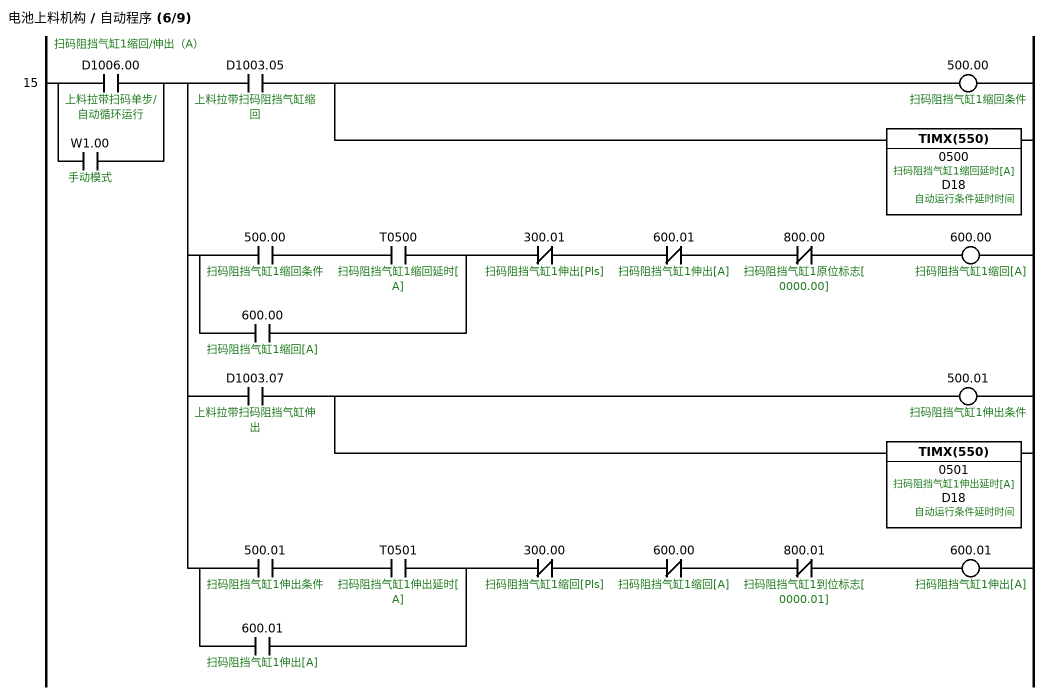
; [picture p24: 电池上料机构 / 自动程序, rungs 15-15]
; rung 15: 扫码阻挡气缸1缩回/伸出（A）
LD D1006.00  ; 上料拉带扫码单步/自动循环运行
OR W1.00  ; 手动模式
OUT TR0
AND D1003.05  ; 上料拉带扫码阻挡气缸缩回
OUT 500.00  ; 扫码阻挡气缸1缩回条件
TIMX(550) 0500 D18  ; 自动运行条件延时时间, 扫码阻挡气缸1缩回延时[A]
LD TR0
LD 500.00  ; 扫码阻挡气缸1缩回条件
AND T0500  ; 扫码阻挡气缸1缩回延时[A]
OR 600.00  ; 扫码阻挡气缸1缩回[A]
ANDLD
ANDNOT 300.01  ; 扫码阻挡气缸1伸出[Pls]
ANDNOT 600.01  ; 扫码阻挡气缸1伸出[A]
ANDNOT 800.00  ; 扫码阻挡气缸1原位标志[0000.00]
OUT 600.00  ; 扫码阻挡气缸1缩回[A]
LD TR0
AND D1003.07  ; 上料拉带扫码阻挡气缸伸出
OUT 500.01  ; 扫码阻挡气缸1伸出条件
TIMX(550) 0501 D18  ; 自动运行条件延时时间, 扫码阻挡气缸1伸出延时[A]
LD TR0
LD 500.01  ; 扫码阻挡气缸1伸出条件
AND T0501  ; 扫码阻挡气缸1伸出延时[A]
OR 600.01  ; 扫码阻挡气缸1伸出[A]
ANDLD
ANDNOT 300.00  ; 扫码阻挡气缸1缩回[Pls]
ANDNOT 600.00  ; 扫码阻挡气缸1缩回[A]
ANDNOT 800.01  ; 扫码阻挡气缸1到位标志[0000.01]
OUT 600.01  ; 扫码阻挡气缸1伸出[A]

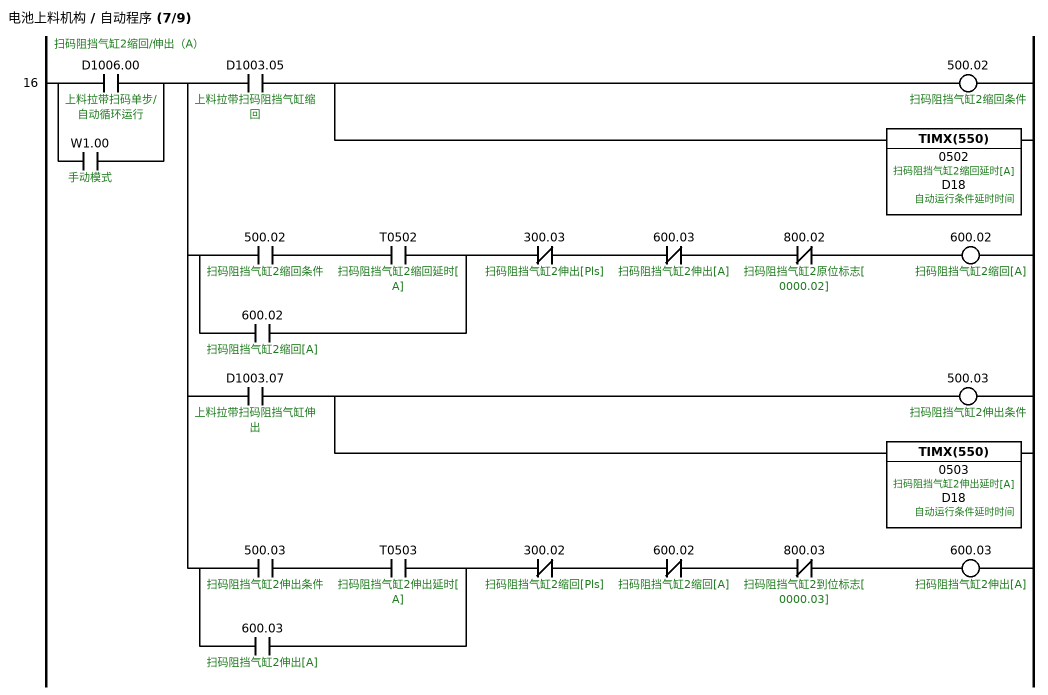
; rung 16: 扫码阻挡气缸2缩回/伸出（A）
LD D1006.00  ; 上料拉带扫码单步/自动循环运行
OR W1.00  ; 手动模式
OUT TR0
AND D1003.05  ; 上料拉带扫码阻挡气缸缩回
OUT 500.02  ; 扫码阻挡气缸2缩回条件
TIMX(550) 0502 D18  ; 自动运行条件延时时间, 扫码阻挡气缸2缩回延时[A]
LD TR0
LD 500.02  ; 扫码阻挡气缸2缩回条件
AND T0502  ; 扫码阻挡气缸2缩回延时[A]
OR 600.02  ; 扫码阻挡气缸2缩回[A]
ANDLD
ANDNOT 300.03  ; 扫码阻挡气缸2伸出[Pls]
ANDNOT 600.03  ; 扫码阻挡气缸2伸出[A]
ANDNOT 800.02  ; 扫码阻挡气缸2原位标志[0000.02]
OUT 600.02  ; 扫码阻挡气缸2缩回[A]
LD TR0
AND D1003.07  ; 上料拉带扫码阻挡气缸伸出
OUT 500.03  ; 扫码阻挡气缸2伸出条件
TIMX(550) 0503 D18  ; 自动运行条件延时时间, 扫码阻挡气缸2伸出延时[A]
LD TR0
LD 500.03  ; 扫码阻挡气缸2伸出条件
AND T0503  ; 扫码阻挡气缸2伸出延时[A]
OR 600.03  ; 扫码阻挡气缸2伸出[A]
ANDLD
ANDNOT 300.02  ; 扫码阻挡气缸2缩回[Pls]
ANDNOT 600.02  ; 扫码阻挡气缸2缩回[A]
ANDNOT 800.03  ; 扫码阻挡气缸2到位标志[0000.03]
OUT 600.03  ; 扫码阻挡气缸2伸出[A]

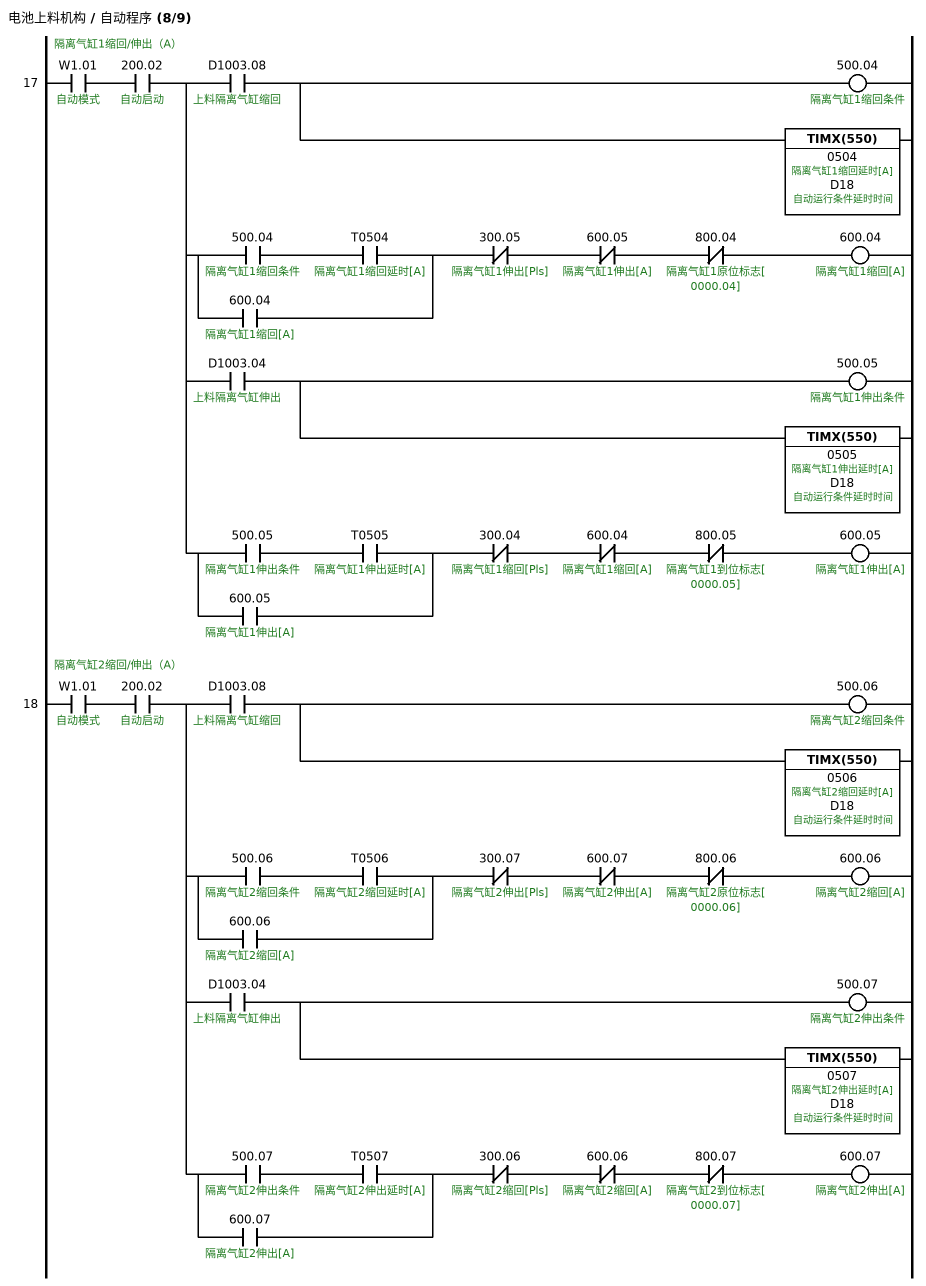
; rung 17: 隔离气缸1缩回/伸出（A）
LD W1.01  ; 自动模式
AND 200.02  ; 自动启动
OUT TR0
AND D1003.08  ; 上料隔离气缸缩回
OUT 500.04  ; 隔离气缸1缩回条件
TIMX(550) 0504 D18  ; 自动运行条件延时时间, 隔离气缸1缩回延时[A]
LD TR0
LD 500.04  ; 隔离气缸1缩回条件
AND T0504  ; 隔离气缸1缩回延时[A]
OR 600.04  ; 隔离气缸1缩回[A]
ANDLD
ANDNOT 300.05  ; 隔离气缸1伸出[Pls]
ANDNOT 600.05  ; 隔离气缸1伸出[A]
ANDNOT 800.04  ; 隔离气缸1原位标志[0000.04]
OUT 600.04  ; 隔离气缸1缩回[A]
LD TR0
AND D1003.04  ; 上料隔离气缸伸出
OUT 500.05  ; 隔离气缸1伸出条件
TIMX(550) 0505 D18  ; 自动运行条件延时时间, 隔离气缸1伸出延时[A]
LD TR0
LD 500.05  ; 隔离气缸1伸出条件
AND T0505  ; 隔离气缸1伸出延时[A]
OR 600.05  ; 隔离气缸1伸出[A]
ANDLD
ANDNOT 300.04  ; 隔离气缸1缩回[Pls]
ANDNOT 600.04  ; 隔离气缸1缩回[A]
ANDNOT 800.05  ; 隔离气缸1到位标志[0000.05]
OUT 600.05  ; 隔离气缸1伸出[A]
; rung 18: 隔离气缸2缩回/伸出（A）
LD W1.01  ; 自动模式
AND 200.02  ; 自动启动
OUT TR0
AND D1003.08  ; 上料隔离气缸缩回
OUT 500.06  ; 隔离气缸2缩回条件
TIMX(550) 0506 D18  ; 自动运行条件延时时间, 隔离气缸2缩回延时[A]
LD TR0
LD 500.06  ; 隔离气缸2缩回条件
AND T0506  ; 隔离气缸2缩回延时[A]
OR 600.06  ; 隔离气缸2缩回[A]
ANDLD
ANDNOT 300.07  ; 隔离气缸2伸出[Pls]
ANDNOT 600.07  ; 隔离气缸2伸出[A]
ANDNOT 800.06  ; 隔离气缸2原位标志[0000.06]
OUT 600.06  ; 隔离气缸2缩回[A]
LD TR0
AND D1003.04  ; 上料隔离气缸伸出
OUT 500.07  ; 隔离气缸2伸出条件
TIMX(550) 0507 D18  ; 自动运行条件延时时间, 隔离气缸2伸出延时[A]
LD TR0
LD 500.07  ; 隔离气缸2伸出条件
AND T0507  ; 隔离气缸2伸出延时[A]
OR 600.07  ; 隔离气缸2伸出[A]
ANDLD
ANDNOT 300.06  ; 隔离气缸2缩回[Pls]
ANDNOT 600.06  ; 隔离气缸2缩回[A]
ANDNOT 800.07  ; 隔离气缸2到位标志[0000.07]
OUT 600.07  ; 隔离气缸2伸出[A]

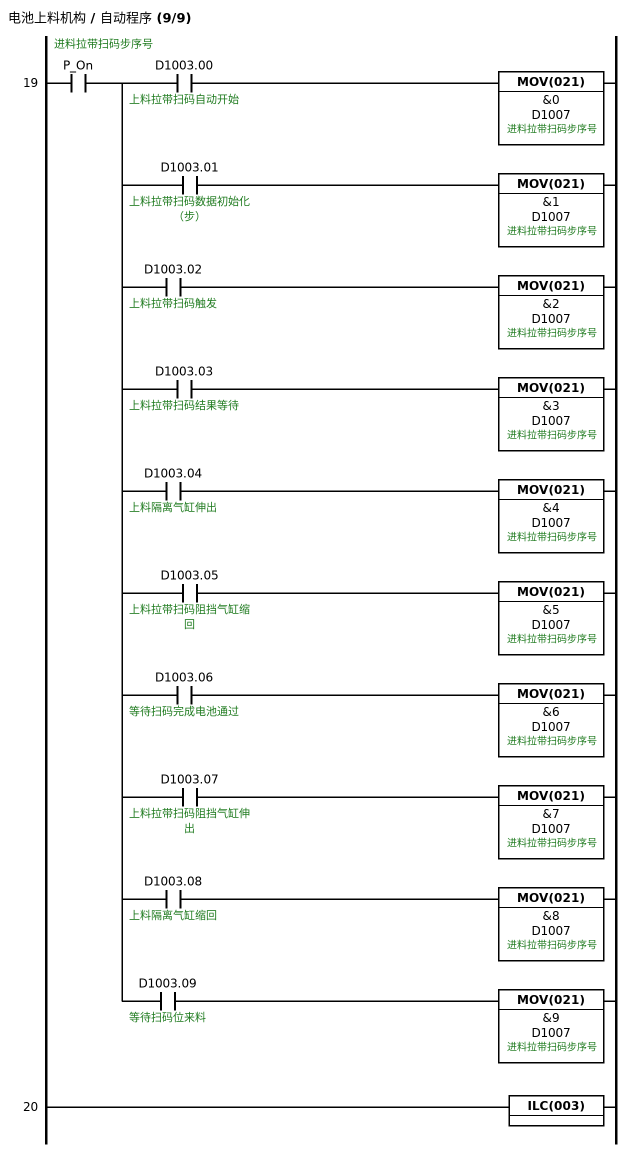
; rung 19: 进料拉带扫码步序号
LD P_On
OUT TR0
AND D1003.00  ; 上料拉带扫码自动开始
MOV(021) &0 D1007  ; 进料拉带扫码步序号
LD TR0
AND D1003.01  ; 上料拉带扫码数据初始化（步）
MOV(021) &1 D1007  ; 进料拉带扫码步序号
LD TR0
AND D1003.02  ; 上料拉带扫码触发
MOV(021) &2 D1007  ; 进料拉带扫码步序号
LD TR0
AND D1003.03  ; 上料拉带扫码结果等待
MOV(021) &3 D1007  ; 进料拉带扫码步序号
LD TR0
AND D1003.04  ; 上料隔离气缸伸出
MOV(021) &4 D1007  ; 进料拉带扫码步序号
LD TR0
AND D1003.05  ; 上料拉带扫码阻挡气缸缩回
MOV(021) &5 D1007  ; 进料拉带扫码步序号
LD TR0
AND D1003.06  ; 等待扫码完成电池通过
MOV(021) &6 D1007  ; 进料拉带扫码步序号
LD TR0
AND D1003.07  ; 上料拉带扫码阻挡气缸伸出
MOV(021) &7 D1007  ; 进料拉带扫码步序号
LD TR0
AND D1003.08  ; 上料隔离气缸缩回
MOV(021) &8 D1007  ; 进料拉带扫码步序号
LD TR0
AND D1003.09  ; 等待扫码位来料
MOV(021) &9 D1007  ; 进料拉带扫码步序号
; rung 20
ILC(003)

### Section 状态指示灯

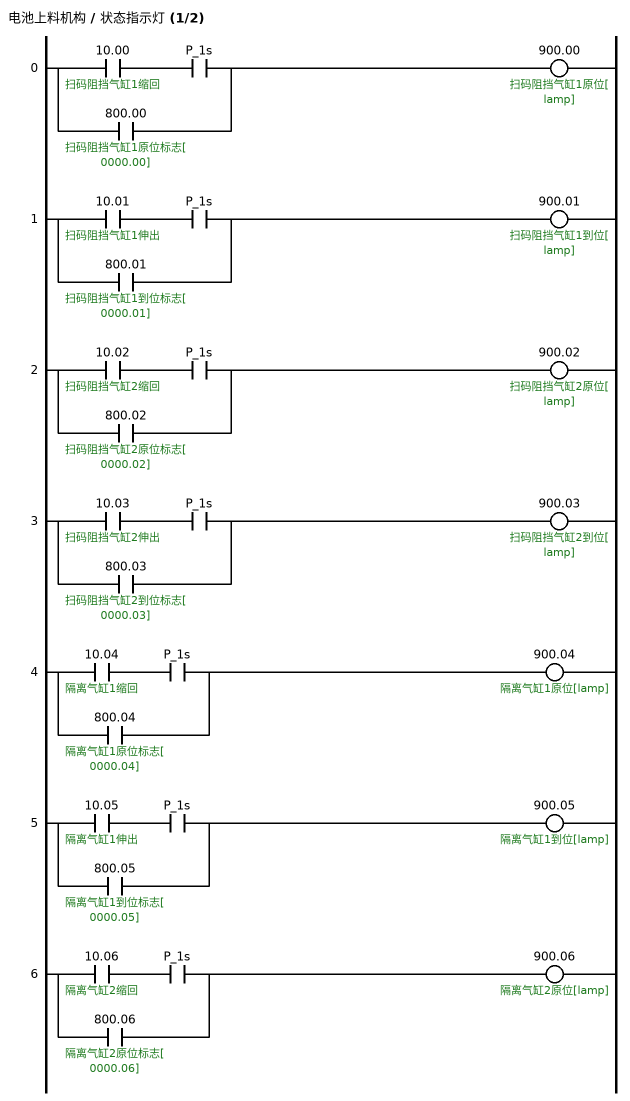
; rung 0
LD 10.00  ; 扫码阻挡气缸1缩回
AND P_1s
OR 800.00  ; 扫码阻挡气缸1原位标志[0000.00]
OUT 900.00  ; 扫码阻挡气缸1原位[lamp]
; rung 1
LD 10.01  ; 扫码阻挡气缸1伸出
AND P_1s
OR 800.01  ; 扫码阻挡气缸1到位标志[0000.01]
OUT 900.01  ; 扫码阻挡气缸1到位[lamp]
; rung 2
LD 10.02  ; 扫码阻挡气缸2缩回
AND P_1s
OR 800.02  ; 扫码阻挡气缸2原位标志[0000.02]
OUT 900.02  ; 扫码阻挡气缸2原位[lamp]
; rung 3
LD 10.03  ; 扫码阻挡气缸2伸出
AND P_1s
OR 800.03  ; 扫码阻挡气缸2到位标志[0000.03]
OUT 900.03  ; 扫码阻挡气缸2到位[lamp]
; rung 4
LD 10.04  ; 隔离气缸1缩回
AND P_1s
OR 800.04  ; 隔离气缸1原位标志[0000.04]
OUT 900.04  ; 隔离气缸1原位[lamp]
; rung 5
LD 10.05  ; 隔离气缸1伸出
AND P_1s
OR 800.05  ; 隔离气缸1到位标志[0000.05]
OUT 900.05  ; 隔离气缸1到位[lamp]
; rung 6
LD 10.06  ; 隔离气缸2缩回
AND P_1s
OR 800.06  ; 隔离气缸2原位标志[0000.06]
OUT 900.06  ; 隔离气缸2原位[lamp]

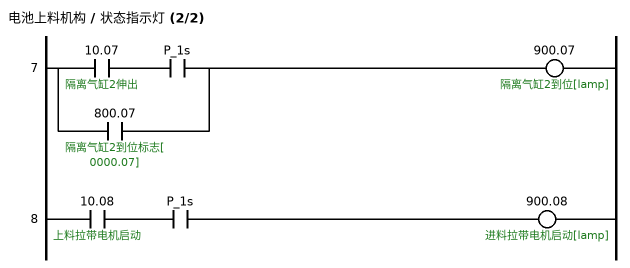
; rung 7
LD 10.07  ; 隔离气缸2伸出
AND P_1s
OR 800.07  ; 隔离气缸2到位标志[0000.07]
OUT 900.07  ; 隔离气缸2到位[lamp]
; rung 8
LD 10.08  ; 上料拉带电机启动
AND P_1s
OUT 900.08  ; 进料拉带电机启动[lamp]

### Section 输出程序

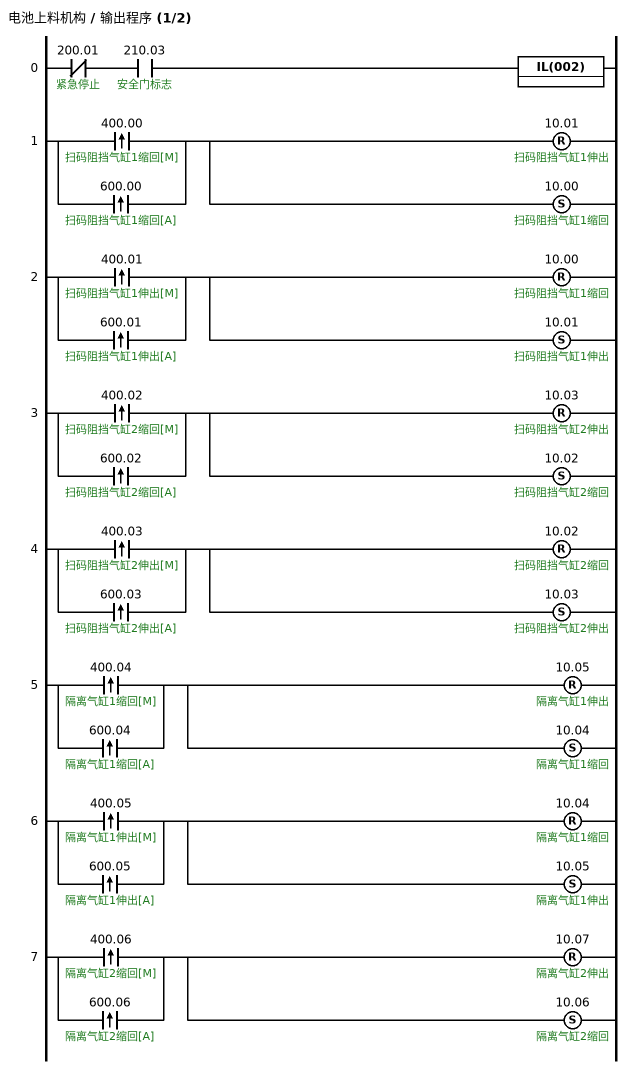
; rung 0
LDNOT 200.01  ; 紧急停止
AND 210.03  ; 安全门标志
IL(002)
; rung 1
@LD 400.00  ; 扫码阻挡气缸1缩回[M]
@OR 600.00  ; 扫码阻挡气缸1缩回[A]
RSET 10.01  ; 扫码阻挡气缸1伸出
SET 10.00  ; 扫码阻挡气缸1缩回
; rung 2
@LD 400.01  ; 扫码阻挡气缸1伸出[M]
@OR 600.01  ; 扫码阻挡气缸1伸出[A]
RSET 10.00  ; 扫码阻挡气缸1缩回
SET 10.01  ; 扫码阻挡气缸1伸出
; rung 3
@LD 400.02  ; 扫码阻挡气缸2缩回[M]
@OR 600.02  ; 扫码阻挡气缸2缩回[A]
RSET 10.03  ; 扫码阻挡气缸2伸出
SET 10.02  ; 扫码阻挡气缸2缩回
; rung 4
@LD 400.03  ; 扫码阻挡气缸2伸出[M]
@OR 600.03  ; 扫码阻挡气缸2伸出[A]
RSET 10.02  ; 扫码阻挡气缸2缩回
SET 10.03  ; 扫码阻挡气缸2伸出
; rung 5
@LD 400.04  ; 隔离气缸1缩回[M]
@OR 600.04  ; 隔离气缸1缩回[A]
RSET 10.05  ; 隔离气缸1伸出
SET 10.04  ; 隔离气缸1缩回
; rung 6
@LD 400.05  ; 隔离气缸1伸出[M]
@OR 600.05  ; 隔离气缸1伸出[A]
RSET 10.04  ; 隔离气缸1缩回
SET 10.05  ; 隔离气缸1伸出
; rung 7
@LD 400.06  ; 隔离气缸2缩回[M]
@OR 600.06  ; 隔离气缸2缩回[A]
RSET 10.07  ; 隔离气缸2伸出
SET 10.06  ; 隔离气缸2缩回

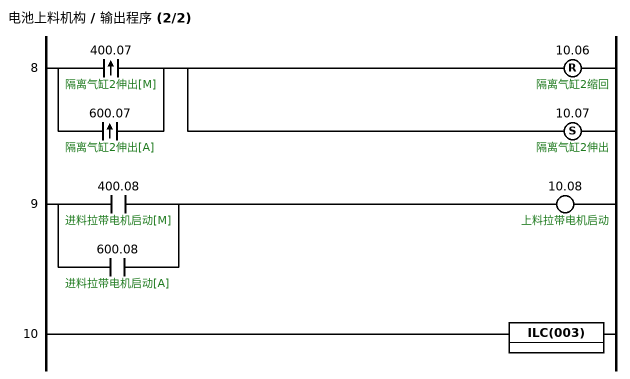
; rung 8
@LD 400.07  ; 隔离气缸2伸出[M]
@OR 600.07  ; 隔离气缸2伸出[A]
RSET 10.06  ; 隔离气缸2缩回
SET 10.07  ; 隔离气缸2伸出
; rung 9
LD 400.08  ; 进料拉带电机启动[M]
OR 600.08  ; 进料拉带电机启动[A]
OUT 10.08  ; 上料拉带电机启动
; rung 10
ILC(003)

### Section END
; rung 0
END(001)

## Program 扫码NG抓取机构 (cyclic task 2)

### Section 主程序

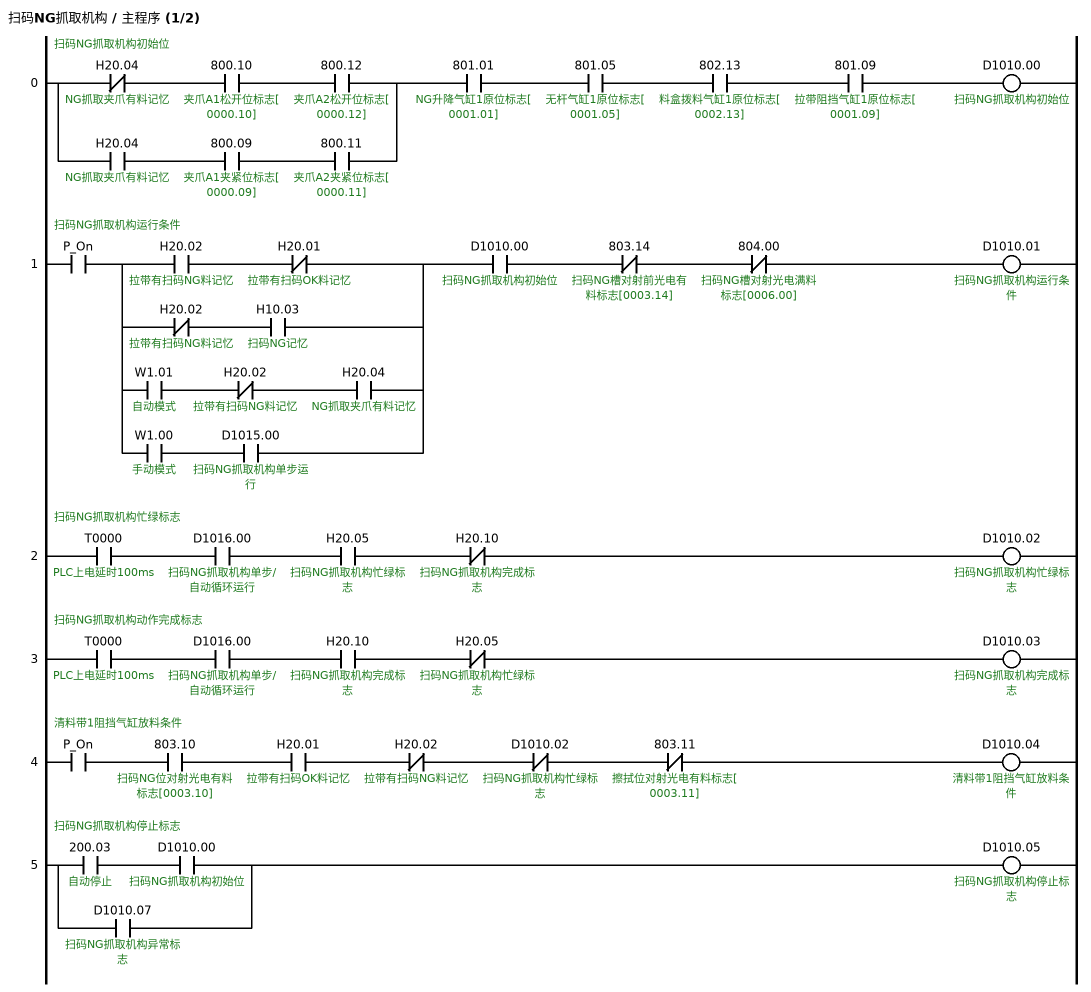
; rung 0: 扫码NG抓取机构初始位
LDNOT H20.04  ; NG抓取夹爪有料记忆
AND 800.10  ; 夹爪A1松开位标志[0000.10]
AND 800.12  ; 夹爪A2松开位标志[0000.12]
LD H20.04  ; NG抓取夹爪有料记忆
AND 800.09  ; 夹爪A1夹紧位标志[0000.09]
AND 800.11  ; 夹爪A2夹紧位标志[0000.11]
ORLD
AND 801.01  ; NG升降气缸1原位标志[0001.01]
AND 801.05  ; 无杆气缸1原位标志[0001.05]
AND 802.13  ; 料盒拨料气缸1原位标志[0002.13]
AND 801.09  ; 拉带阻挡气缸1原位标志[0001.09]
OUT D1010.00  ; 扫码NG抓取机构初始位
; rung 1: 扫码NG抓取机构运行条件
LD P_On
LD H20.02  ; 拉带有扫码NG料记忆
ANDNOT H20.01  ; 拉带有扫码OK料记忆
LDNOT H20.02  ; 拉带有扫码NG料记忆
AND H10.03  ; 扫码NG记忆
ORLD
LD W1.01  ; 自动模式
ANDNOT H20.02  ; 拉带有扫码NG料记忆
AND H20.04  ; NG抓取夹爪有料记忆
ORLD
LD W1.00  ; 手动模式
AND D1015.00  ; 扫码NG抓取机构单步运行
ORLD
ANDLD
AND D1010.00  ; 扫码NG抓取机构初始位
ANDNOT 803.14  ; 扫码NG槽对射前光电有料标志[0003.14]
ANDNOT 804.00  ; 扫码NG槽对射光电满料标志[0006.00]
OUT D1010.01  ; 扫码NG抓取机构运行条件
; rung 2: 扫码NG抓取机构忙绿标志
LD T0000  ; PLC上电延时100ms
AND D1016.00  ; 扫码NG抓取机构单步/自动循环运行
AND H20.05  ; 扫码NG抓取机构忙绿标志
ANDNOT H20.10  ; 扫码NG抓取机构完成标志
OUT D1010.02  ; 扫码NG抓取机构忙绿标志
; rung 3: 扫码NG抓取机构动作完成标志
LD T0000  ; PLC上电延时100ms
AND D1016.00  ; 扫码NG抓取机构单步/自动循环运行
AND H20.10  ; 扫码NG抓取机构完成标志
ANDNOT H20.05  ; 扫码NG抓取机构忙绿标志
OUT D1010.03  ; 扫码NG抓取机构完成标志
; rung 4: 清料带1阻挡气缸放料条件
LD P_On
AND 803.10  ; 扫码NG位对射光电有料标志[0003.10]
AND H20.01  ; 拉带有扫码OK料记忆
ANDNOT H20.02  ; 拉带有扫码NG料记忆
ANDNOT D1010.02  ; 扫码NG抓取机构忙绿标志
ANDNOT 803.11  ; 擦拭位对射光电有料标志[0003.11]
OUT D1010.04  ; 清料带1阻挡气缸放料条件
; rung 5: 扫码NG抓取机构停止标志
LD 200.03  ; 自动停止
AND D1010.00  ; 扫码NG抓取机构初始位
OR D1010.07  ; 扫码NG抓取机构异常标志
OUT D1010.05  ; 扫码NG抓取机构停止标志

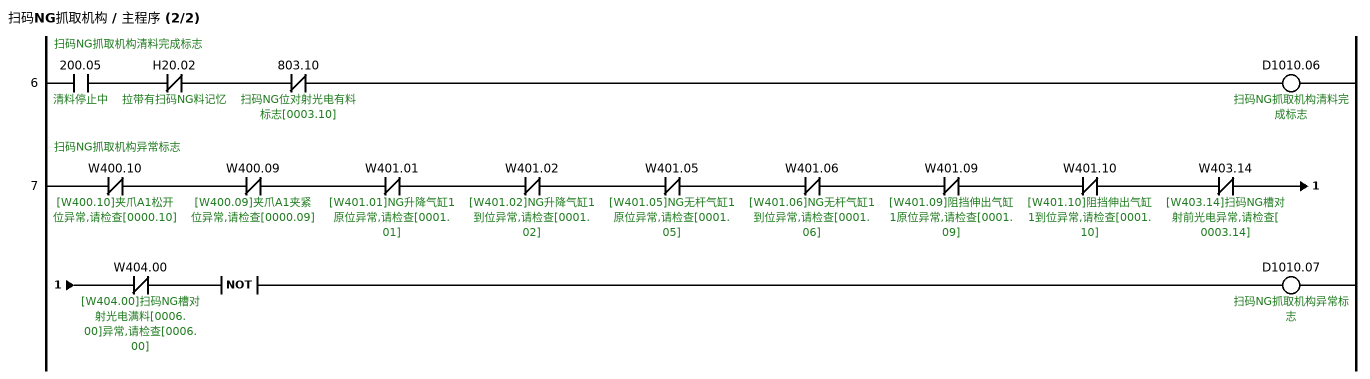
; rung 6: 扫码NG抓取机构清料完成标志
LD 200.05  ; 清料停止中
ANDNOT H20.02  ; 拉带有扫码NG料记忆
ANDNOT 803.10  ; 扫码NG位对射光电有料标志[0003.10]
OUT D1010.06  ; 扫码NG抓取机构清料完成标志
; rung 7: 扫码NG抓取机构异常标志
LDNOT W400.10  ; [W400.10]夹爪A1松开位异常,请检查[0000.10]
ANDNOT W400.09  ; [W400.09]夹爪A1夹紧位异常,请检查[0000.09]
ANDNOT W401.01  ; [W401.01]NG升降气缸1原位异常,请检查[0001.01]
ANDNOT W401.02  ; [W401.02]NG升降气缸1到位异常,请检查[0001.02]
ANDNOT W401.05  ; [W401.05]NG无杆气缸1原位异常,请检查[0001.05]
ANDNOT W401.06  ; [W401.06]NG无杆气缸1到位异常,请检查[0001.06]
ANDNOT W401.09  ; [W401.09]阻挡伸出气缸1原位异常,请检查[0001.09]
ANDNOT W401.10  ; [W401.10]阻挡伸出气缸1到位异常,请检查[0001.10]
ANDNOT W403.14  ; [W403.14]扫码NG槽对射前光电异常,请检查[0003.14]
ANDNOT W404.00  ; [W404.00]扫码NG槽对射光电满料[0006.00]异常,请检查[0006.00]
NOT(520)
OUT D1010.07  ; 扫码NG抓取机构异常标志

### Section 工站复位

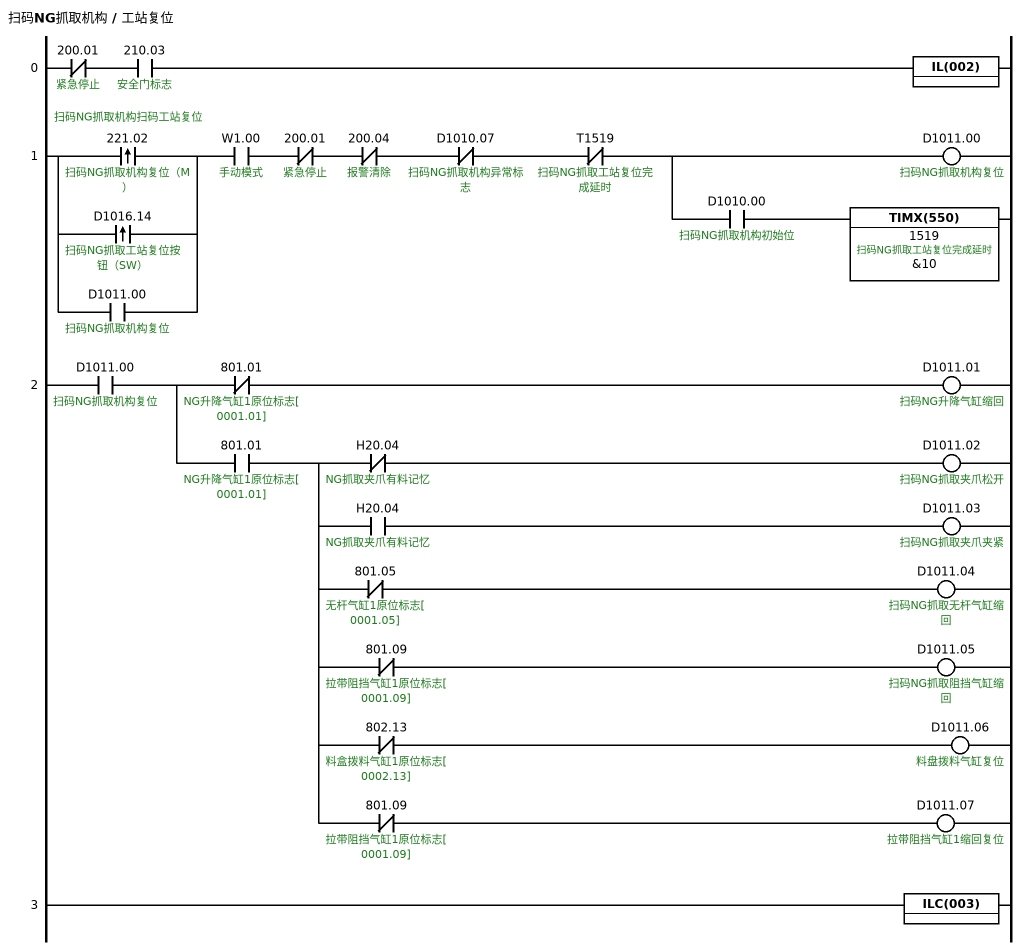
; rung 0
LDNOT 200.01  ; 紧急停止
AND 210.03  ; 安全门标志
IL(002)
; rung 1: 扫码NG抓取机构扫码工站复位
@LD 221.02  ; 扫码NG抓取机构复位（M）
@OR D1016.14  ; 扫码NG抓取工站复位按钮（SW）
OR D1011.00  ; 扫码NG抓取机构复位
AND W1.00  ; 手动模式
ANDNOT 200.01  ; 紧急停止
ANDNOT 200.04  ; 报警清除
ANDNOT D1010.07  ; 扫码NG抓取机构异常标志
ANDNOT T1519  ; 扫码NG抓取工站复位完成延时
OUT D1011.00  ; 扫码NG抓取机构复位
AND D1010.00  ; 扫码NG抓取机构初始位
TIMX(550) 1519 &10  ; 扫码NG抓取工站复位完成延时
; rung 2
LD D1011.00  ; 扫码NG抓取机构复位
OUT TR0
ANDNOT 801.01  ; NG升降气缸1原位标志[0001.01]
OUT D1011.01  ; 扫码NG升降气缸缩回
LD TR0
AND 801.01  ; NG升降气缸1原位标志[0001.01]
OUT TR0
ANDNOT H20.04  ; NG抓取夹爪有料记忆
OUT D1011.02  ; 扫码NG抓取夹爪松开
LD TR0
AND H20.04  ; NG抓取夹爪有料记忆
OUT D1011.03  ; 扫码NG抓取夹爪夹紧
LD TR0
ANDNOT 801.05  ; 无杆气缸1原位标志[0001.05]
OUT D1011.04  ; 扫码NG抓取无杆气缸缩回
LD TR0
ANDNOT 801.09  ; 拉带阻挡气缸1原位标志[0001.09]
OUT D1011.05  ; 扫码NG抓取阻挡气缸缩回
LD TR0
ANDNOT 802.13  ; 料盒拨料气缸1原位标志[0002.13]
OUT D1011.06  ; 料盘拨料气缸复位
LD TR0
ANDNOT 801.09  ; 拉带阻挡气缸1原位标志[0001.09]
OUT D1011.07  ; 拉带阻挡气缸1缩回复位
; rung 3
ILC(003)

### Section 手动程序

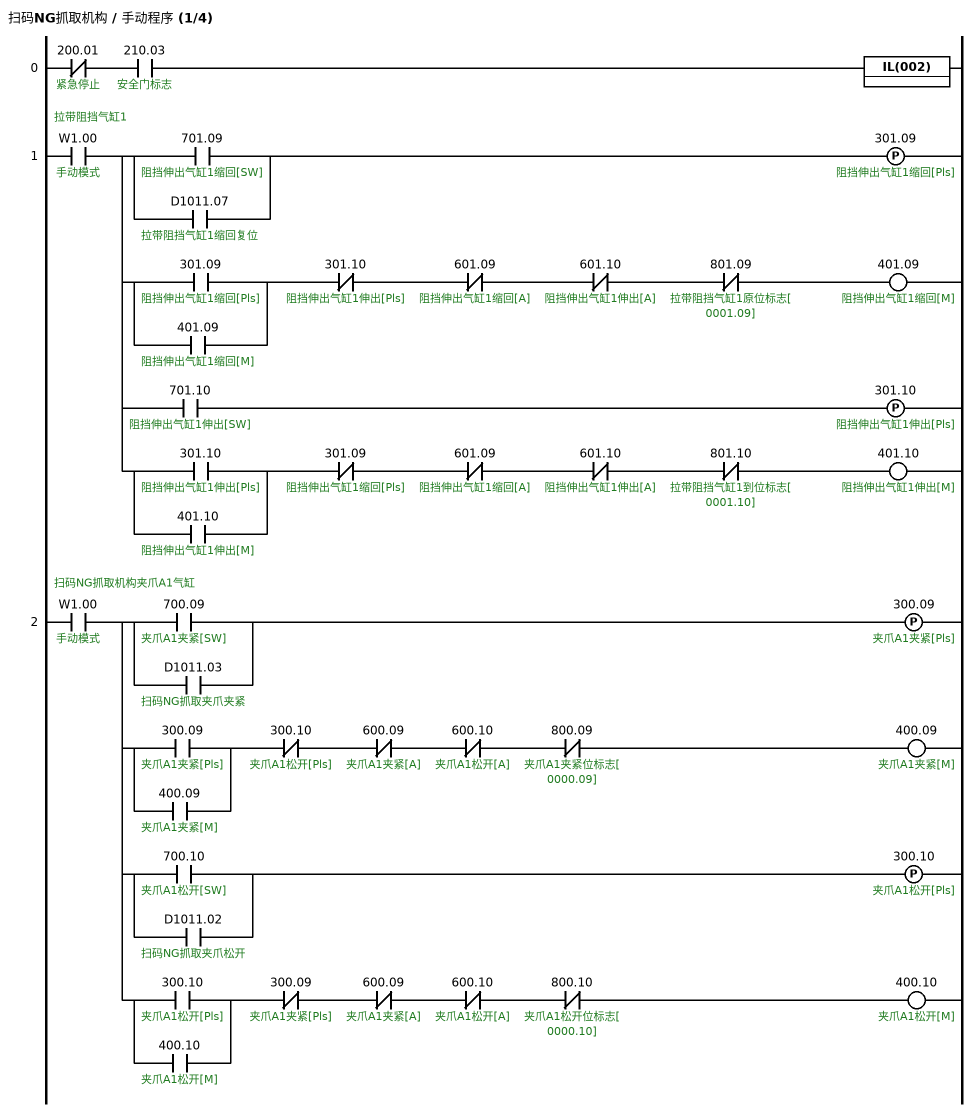
; rung 0
LDNOT 200.01  ; 紧急停止
AND 210.03  ; 安全门标志
IL(002)
; rung 1: 拉带阻挡气缸1
LD W1.00  ; 手动模式
OUT TR0
LD 701.09  ; 阻挡伸出气缸1缩回[SW]
OR D1011.07  ; 拉带阻挡气缸1缩回复位
ANDLD
DIFU(013) 301.09  ; 阻挡伸出气缸1缩回[Pls]
LD TR0
LD 301.09  ; 阻挡伸出气缸1缩回[Pls]
OR 401.09  ; 阻挡伸出气缸1缩回[M]
ANDLD
ANDNOT 301.10  ; 阻挡伸出气缸1伸出[Pls]
ANDNOT 601.09  ; 阻挡伸出气缸1缩回[A]
ANDNOT 601.10  ; 阻挡伸出气缸1伸出[A]
ANDNOT 801.09  ; 拉带阻挡气缸1原位标志[0001.09]
OUT 401.09  ; 阻挡伸出气缸1缩回[M]
LD TR0
AND 701.10  ; 阻挡伸出气缸1伸出[SW]
DIFU(013) 301.10  ; 阻挡伸出气缸1伸出[Pls]
LD TR0
LD 301.10  ; 阻挡伸出气缸1伸出[Pls]
OR 401.10  ; 阻挡伸出气缸1伸出[M]
ANDLD
ANDNOT 301.09  ; 阻挡伸出气缸1缩回[Pls]
ANDNOT 601.09  ; 阻挡伸出气缸1缩回[A]
ANDNOT 601.10  ; 阻挡伸出气缸1伸出[A]
ANDNOT 801.10  ; 拉带阻挡气缸1到位标志[0001.10]
OUT 401.10  ; 阻挡伸出气缸1伸出[M]
; rung 2: 扫码NG抓取机构夹爪A1气缸
LD W1.00  ; 手动模式
OUT TR0
LD 700.09  ; 夹爪A1夹紧[SW]
OR D1011.03  ; 扫码NG抓取夹爪夹紧
ANDLD
DIFU(013) 300.09  ; 夹爪A1夹紧[Pls]
LD TR0
LD 300.09  ; 夹爪A1夹紧[Pls]
OR 400.09  ; 夹爪A1夹紧[M]
ANDLD
ANDNOT 300.10  ; 夹爪A1松开[Pls]
ANDNOT 600.09  ; 夹爪A1夹紧[A]
ANDNOT 600.10  ; 夹爪A1松开[A]
ANDNOT 800.09  ; 夹爪A1夹紧位标志[0000.09]
OUT 400.09  ; 夹爪A1夹紧[M]
LD TR0
LD 700.10  ; 夹爪A1松开[SW]
OR D1011.02  ; 扫码NG抓取夹爪松开
ANDLD
DIFU(013) 300.10  ; 夹爪A1松开[Pls]
LD TR0
LD 300.10  ; 夹爪A1松开[Pls]
OR 400.10  ; 夹爪A1松开[M]
ANDLD
ANDNOT 300.09  ; 夹爪A1夹紧[Pls]
ANDNOT 600.09  ; 夹爪A1夹紧[A]
ANDNOT 600.10  ; 夹爪A1松开[A]
ANDNOT 800.10  ; 夹爪A1松开位标志[0000.10]
OUT 400.10  ; 夹爪A1松开[M]

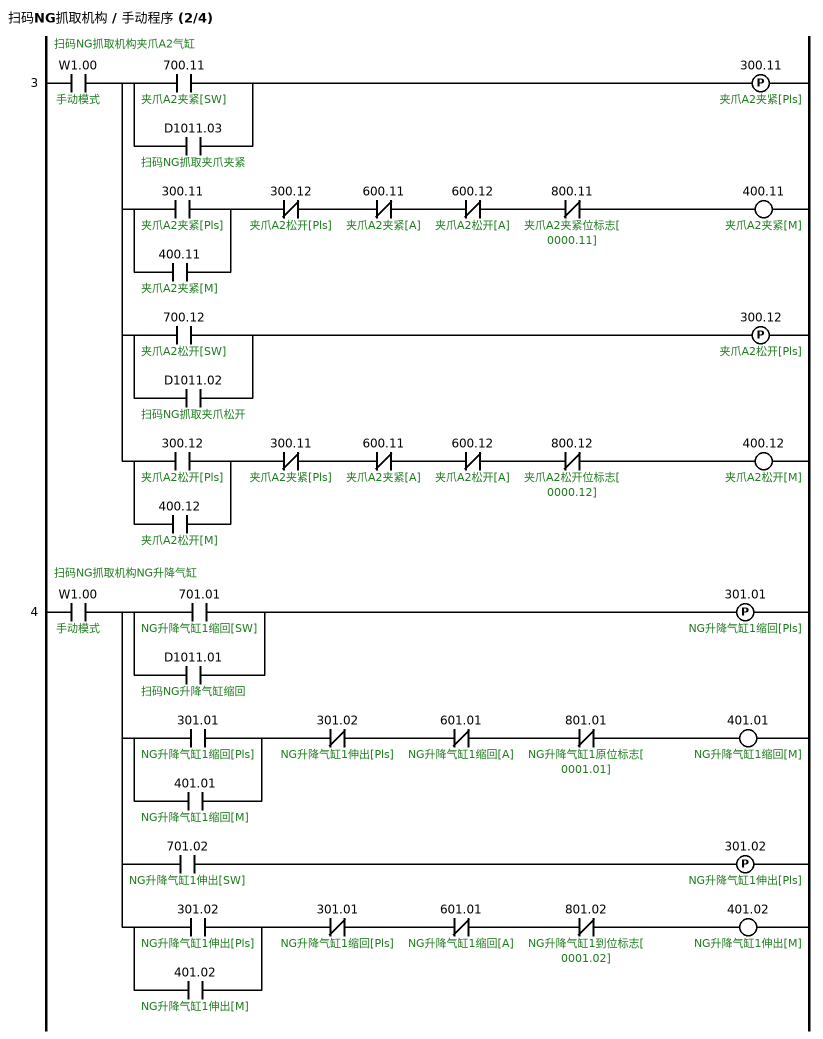
; rung 3: 扫码NG抓取机构夹爪A2气缸
LD W1.00  ; 手动模式
OUT TR0
LD 700.11  ; 夹爪A2夹紧[SW]
OR D1011.03  ; 扫码NG抓取夹爪夹紧
ANDLD
DIFU(013) 300.11  ; 夹爪A2夹紧[Pls]
LD TR0
LD 300.11  ; 夹爪A2夹紧[Pls]
OR 400.11  ; 夹爪A2夹紧[M]
ANDLD
ANDNOT 300.12  ; 夹爪A2松开[Pls]
ANDNOT 600.11  ; 夹爪A2夹紧[A]
ANDNOT 600.12  ; 夹爪A2松开[A]
ANDNOT 800.11  ; 夹爪A2夹紧位标志[0000.11]
OUT 400.11  ; 夹爪A2夹紧[M]
LD TR0
LD 700.12  ; 夹爪A2松开[SW]
OR D1011.02  ; 扫码NG抓取夹爪松开
ANDLD
DIFU(013) 300.12  ; 夹爪A2松开[Pls]
LD TR0
LD 300.12  ; 夹爪A2松开[Pls]
OR 400.12  ; 夹爪A2松开[M]
ANDLD
ANDNOT 300.11  ; 夹爪A2夹紧[Pls]
ANDNOT 600.11  ; 夹爪A2夹紧[A]
ANDNOT 600.12  ; 夹爪A2松开[A]
ANDNOT 800.12  ; 夹爪A2松开位标志[0000.12]
OUT 400.12  ; 夹爪A2松开[M]
; rung 4: 扫码NG抓取机构NG升降气缸
LD W1.00  ; 手动模式
OUT TR0
LD 701.01  ; NG升降气缸1缩回[SW]
OR D1011.01  ; 扫码NG升降气缸缩回
ANDLD
DIFU(013) 301.01  ; NG升降气缸1缩回[Pls]
LD TR0
LD 301.01  ; NG升降气缸1缩回[Pls]
OR 401.01  ; NG升降气缸1缩回[M]
ANDLD
ANDNOT 301.02  ; NG升降气缸1伸出[Pls]
ANDNOT 601.01  ; NG升降气缸1缩回[A]
ANDNOT 801.01  ; NG升降气缸1原位标志[0001.01]
OUT 401.01  ; NG升降气缸1缩回[M]
LD TR0
AND 701.02  ; NG升降气缸1伸出[SW]
DIFU(013) 301.02  ; NG升降气缸1伸出[Pls]
LD TR0
LD 301.02  ; NG升降气缸1伸出[Pls]
OR 401.02  ; NG升降气缸1伸出[M]
ANDLD
ANDNOT 301.01  ; NG升降气缸1缩回[Pls]
ANDNOT 601.01  ; NG升降气缸1缩回[A]
ANDNOT 801.02  ; NG升降气缸1到位标志[0001.02]
OUT 401.02  ; NG升降气缸1伸出[M]

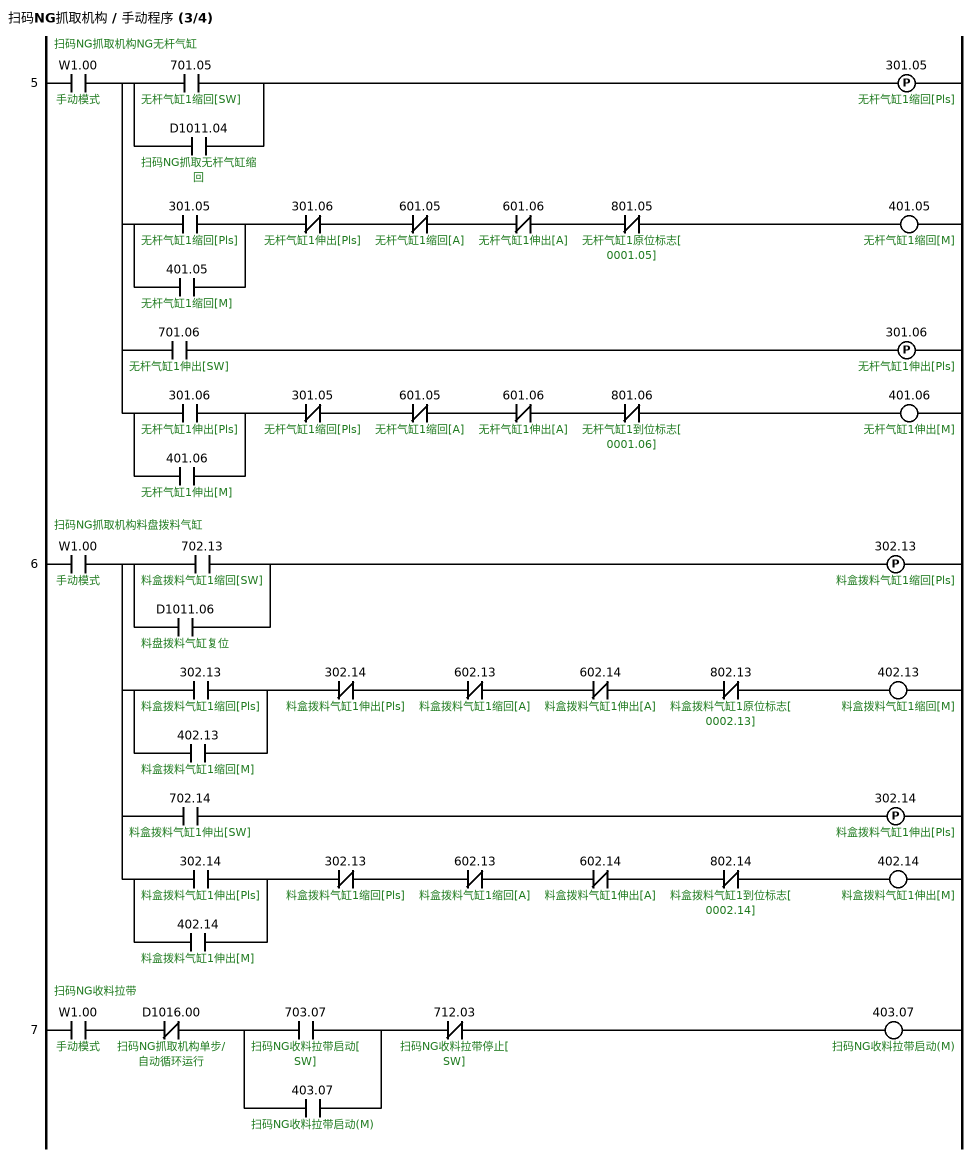
; rung 5: 扫码NG抓取机构NG无杆气缸
LD W1.00  ; 手动模式
OUT TR0
LD 701.05  ; 无杆气缸1缩回[SW]
OR D1011.04  ; 扫码NG抓取无杆气缸缩回
ANDLD
DIFU(013) 301.05  ; 无杆气缸1缩回[Pls]
LD TR0
LD 301.05  ; 无杆气缸1缩回[Pls]
OR 401.05  ; 无杆气缸1缩回[M]
ANDLD
ANDNOT 301.06  ; 无杆气缸1伸出[Pls]
ANDNOT 601.05  ; 无杆气缸1缩回[A]
ANDNOT 601.06  ; 无杆气缸1伸出[A]
ANDNOT 801.05  ; 无杆气缸1原位标志[0001.05]
OUT 401.05  ; 无杆气缸1缩回[M]
LD TR0
AND 701.06  ; 无杆气缸1伸出[SW]
DIFU(013) 301.06  ; 无杆气缸1伸出[Pls]
LD TR0
LD 301.06  ; 无杆气缸1伸出[Pls]
OR 401.06  ; 无杆气缸1伸出[M]
ANDLD
ANDNOT 301.05  ; 无杆气缸1缩回[Pls]
ANDNOT 601.05  ; 无杆气缸1缩回[A]
ANDNOT 601.06  ; 无杆气缸1伸出[A]
ANDNOT 801.06  ; 无杆气缸1到位标志[0001.06]
OUT 401.06  ; 无杆气缸1伸出[M]
; rung 6: 扫码NG抓取机构料盘拨料气缸
LD W1.00  ; 手动模式
OUT TR0
LD 702.13  ; 料盒拨料气缸1缩回[SW]
OR D1011.06  ; 料盘拨料气缸复位
ANDLD
DIFU(013) 302.13  ; 料盒拨料气缸1缩回[Pls]
LD TR0
LD 302.13  ; 料盒拨料气缸1缩回[Pls]
OR 402.13  ; 料盒拨料气缸1缩回[M]
ANDLD
ANDNOT 302.14  ; 料盒拨料气缸1伸出[Pls]
ANDNOT 602.13  ; 料盒拨料气缸1缩回[A]
ANDNOT 602.14  ; 料盒拨料气缸1伸出[A]
ANDNOT 802.13  ; 料盒拨料气缸1原位标志[0002.13]
OUT 402.13  ; 料盒拨料气缸1缩回[M]
LD TR0
AND 702.14  ; 料盒拨料气缸1伸出[SW]
DIFU(013) 302.14  ; 料盒拨料气缸1伸出[Pls]
LD TR0
LD 302.14  ; 料盒拨料气缸1伸出[Pls]
OR 402.14  ; 料盒拨料气缸1伸出[M]
ANDLD
ANDNOT 302.13  ; 料盒拨料气缸1缩回[Pls]
ANDNOT 602.13  ; 料盒拨料气缸1缩回[A]
ANDNOT 602.14  ; 料盒拨料气缸1伸出[A]
ANDNOT 802.14  ; 料盒拨料气缸1到位标志[0002.14]
OUT 402.14  ; 料盒拨料气缸1伸出[M]
; rung 7: 扫码NG收料拉带
LD W1.00  ; 手动模式
ANDNOT D1016.00  ; 扫码NG抓取机构单步/自动循环运行
LD 703.07  ; 扫码NG收料拉带启动[SW]
OR 403.07  ; 扫码NG收料拉带启动(M)
ANDLD
ANDNOT 712.03  ; 扫码NG收料拉带停止[SW]
OUT 403.07  ; 扫码NG收料拉带启动(M)

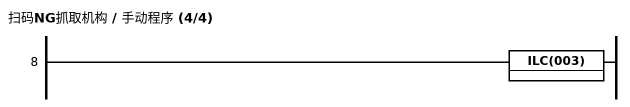
; rung 8
ILC(003)

### Section 自动程序

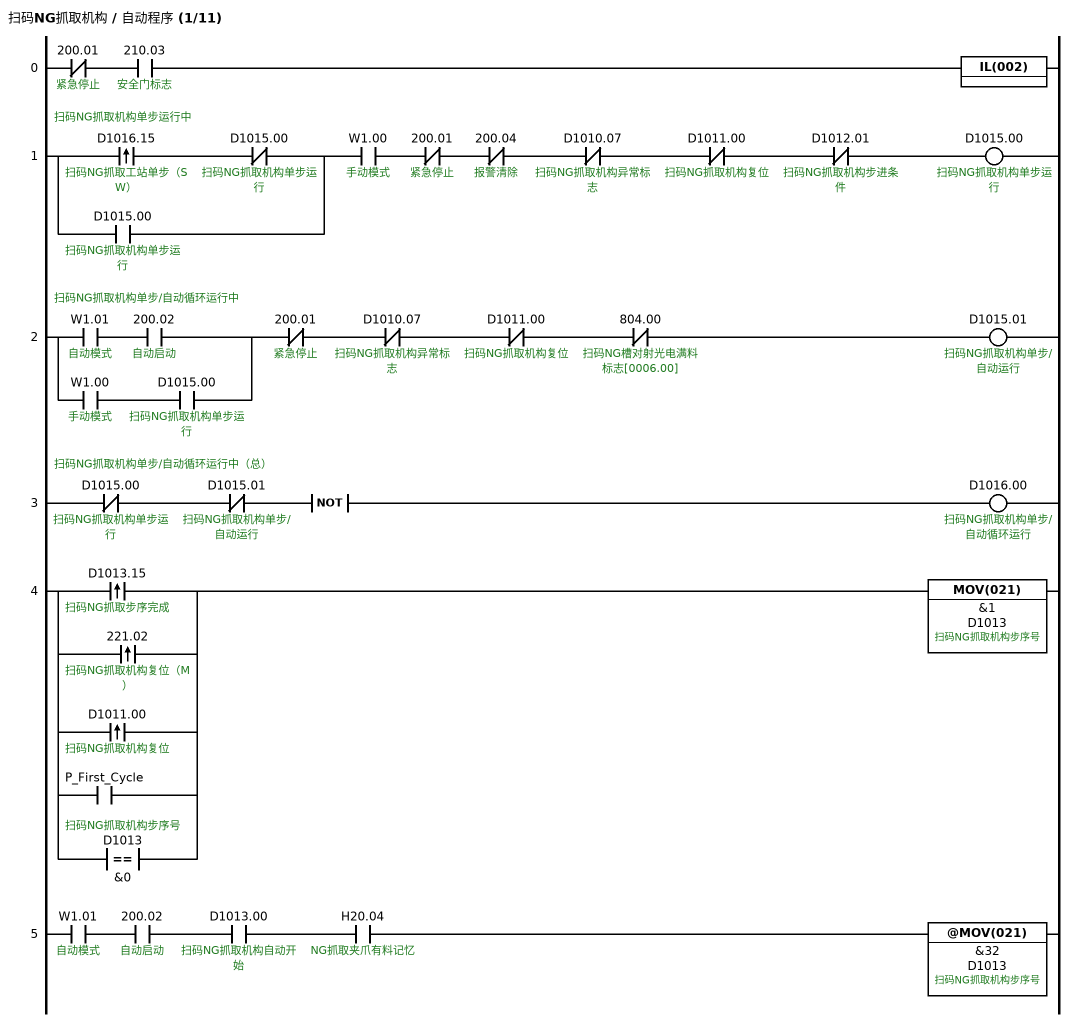
; rung 0
LDNOT 200.01  ; 紧急停止
AND 210.03  ; 安全门标志
IL(002)
; rung 1: 扫码NG抓取机构单步运行中
@LD D1016.15  ; 扫码NG抓取工站单步（SW）
ANDNOT D1015.00  ; 扫码NG抓取机构单步运行
OR D1015.00  ; 扫码NG抓取机构单步运行
AND W1.00  ; 手动模式
ANDNOT 200.01  ; 紧急停止
ANDNOT 200.04  ; 报警清除
ANDNOT D1010.07  ; 扫码NG抓取机构异常标志
ANDNOT D1011.00  ; 扫码NG抓取机构复位
ANDNOT D1012.01  ; 扫码NG抓取机构步进条件
OUT D1015.00  ; 扫码NG抓取机构单步运行
; rung 2: 扫码NG抓取机构单步/自动循环运行中
LD W1.01  ; 自动模式
AND 200.02  ; 自动启动
LD W1.00  ; 手动模式
AND D1015.00  ; 扫码NG抓取机构单步运行
ORLD
ANDNOT 200.01  ; 紧急停止
ANDNOT D1010.07  ; 扫码NG抓取机构异常标志
ANDNOT D1011.00  ; 扫码NG抓取机构复位
ANDNOT 804.00  ; 扫码NG槽对射光电满料标志[0006.00]
OUT D1015.01  ; 扫码NG抓取机构单步/自动运行
; rung 3: 扫码NG抓取机构单步/自动循环运行中（总）
LDNOT D1015.00  ; 扫码NG抓取机构单步运行
ANDNOT D1015.01  ; 扫码NG抓取机构单步/自动运行
NOT(520)
OUT D1016.00  ; 扫码NG抓取机构单步/自动循环运行
; rung 4
@LD D1013.15  ; 扫码NG抓取步序完成
@OR 221.02  ; 扫码NG抓取机构复位（M）
@OR D1011.00  ; 扫码NG抓取机构复位
OR P_First_Cycle
OR=(300) D1013 &0  ; 扫码NG抓取机构步序号
MOV(021) &1 D1013  ; 扫码NG抓取机构步序号
; rung 5
LD W1.01  ; 自动模式
AND 200.02  ; 自动启动
AND D1013.00  ; 扫码NG抓取机构自动开始
AND H20.04  ; NG抓取夹爪有料记忆
@MOV(021) &32 D1013  ; 扫码NG抓取机构步序号

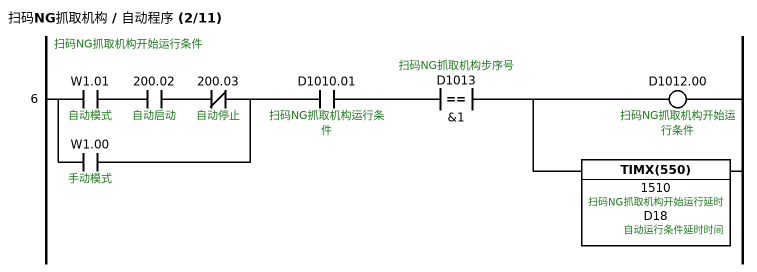
; rung 6: 扫码NG抓取机构开始运行条件
LD W1.01  ; 自动模式
AND 200.02  ; 自动启动
ANDNOT 200.03  ; 自动停止
OR W1.00  ; 手动模式
AND D1010.01  ; 扫码NG抓取机构运行条件
AND=(300) D1013 &1  ; 扫码NG抓取机构步序号
OUT D1012.00  ; 扫码NG抓取机构开始运行条件
TIMX(550) 1510 D18  ; 自动运行条件延时时间, 扫码NG抓取机构开始运行延时

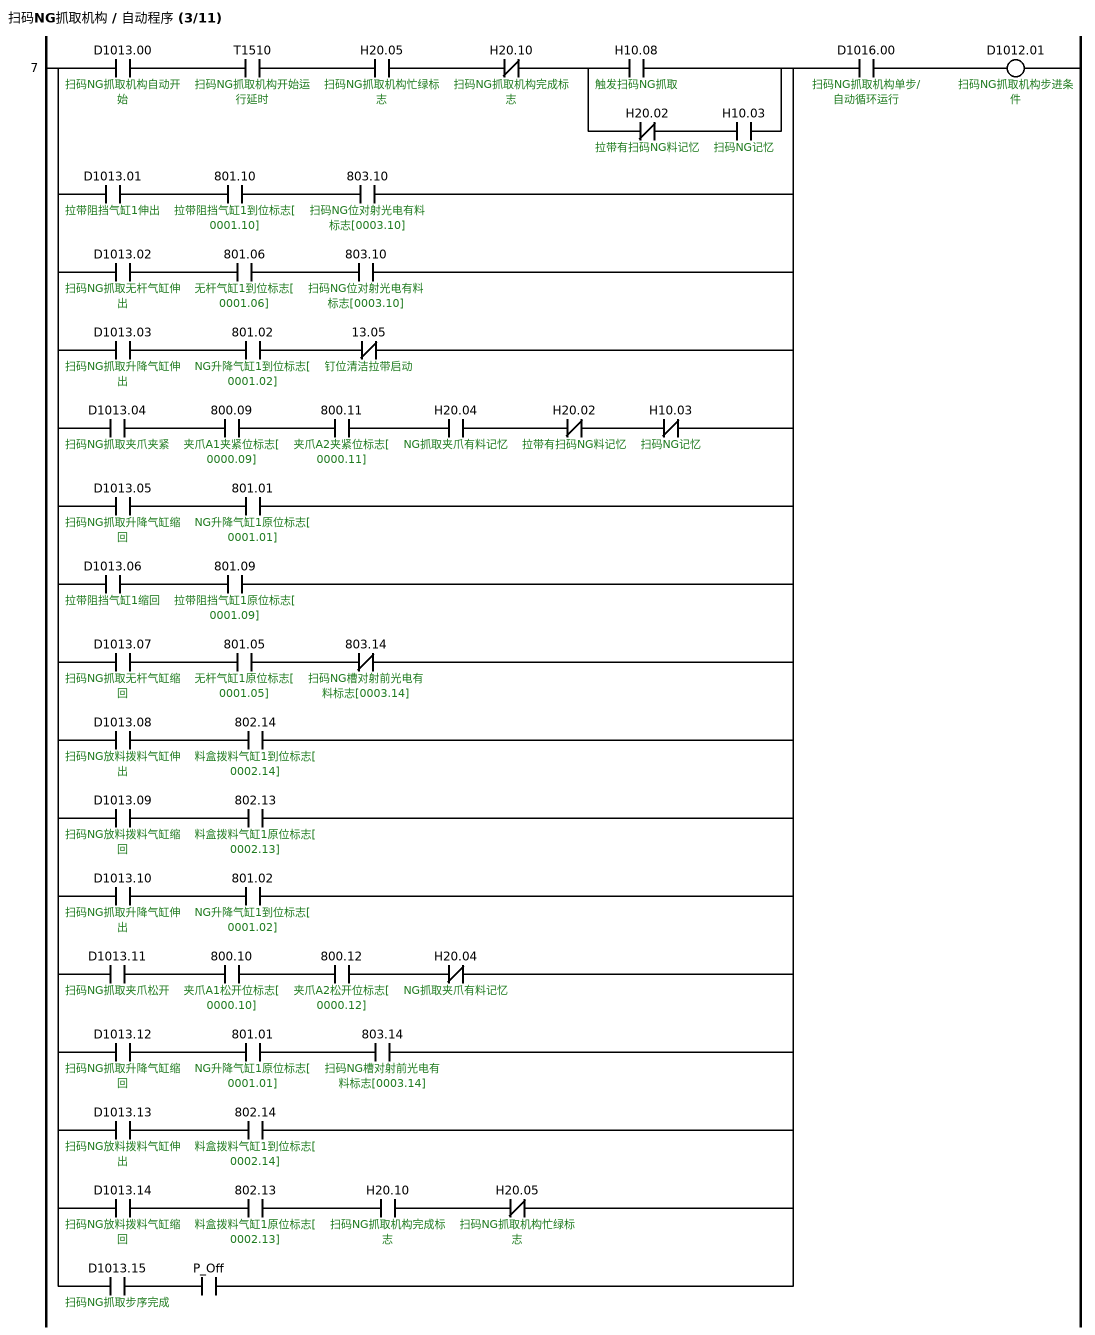
; rung 7
LD D1013.00  ; 扫码NG抓取机构自动开始
AND T1510  ; 扫码NG抓取机构开始运行延时
AND H20.05  ; 扫码NG抓取机构忙绿标志
ANDNOT H20.10  ; 扫码NG抓取机构完成标志
LD H10.08  ; 触发扫码NG抓取
LDNOT H20.02  ; 拉带有扫码NG料记忆
AND H10.03  ; 扫码NG记忆
ORLD
ANDLD
LD D1013.01  ; 拉带阻挡气缸1伸出
AND 801.10  ; 拉带阻挡气缸1到位标志[0001.10]
AND 803.10  ; 扫码NG位对射光电有料标志[0003.10]
ORLD
LD D1013.02  ; 扫码NG抓取无杆气缸伸出
AND 801.06  ; 无杆气缸1到位标志[0001.06]
AND 803.10  ; 扫码NG位对射光电有料标志[0003.10]
ORLD
LD D1013.03  ; 扫码NG抓取升降气缸伸出
AND 801.02  ; NG升降气缸1到位标志[0001.02]
ANDNOT 13.05  ; 钉位清洁拉带启动
ORLD
LD D1013.04  ; 扫码NG抓取夹爪夹紧
AND 800.09  ; 夹爪A1夹紧位标志[0000.09]
AND 800.11  ; 夹爪A2夹紧位标志[0000.11]
AND H20.04  ; NG抓取夹爪有料记忆
ANDNOT H20.02  ; 拉带有扫码NG料记忆
ANDNOT H10.03  ; 扫码NG记忆
ORLD
LD D1013.05  ; 扫码NG抓取升降气缸缩回
AND 801.01  ; NG升降气缸1原位标志[0001.01]
ORLD
LD D1013.06  ; 拉带阻挡气缸1缩回
AND 801.09  ; 拉带阻挡气缸1原位标志[0001.09]
ORLD
LD D1013.07  ; 扫码NG抓取无杆气缸缩回
AND 801.05  ; 无杆气缸1原位标志[0001.05]
ANDNOT 803.14  ; 扫码NG槽对射前光电有料标志[0003.14]
ORLD
LD D1013.08  ; 扫码NG放料拨料气缸伸出
AND 802.14  ; 料盒拨料气缸1到位标志[0002.14]
ORLD
LD D1013.09  ; 扫码NG放料拨料气缸缩回
AND 802.13  ; 料盒拨料气缸1原位标志[0002.13]
ORLD
LD D1013.10  ; 扫码NG抓取升降气缸伸出
AND 801.02  ; NG升降气缸1到位标志[0001.02]
ORLD
LD D1013.11  ; 扫码NG抓取夹爪松开
AND 800.10  ; 夹爪A1松开位标志[0000.10]
AND 800.12  ; 夹爪A2松开位标志[0000.12]
ANDNOT H20.04  ; NG抓取夹爪有料记忆
ORLD
LD D1013.12  ; 扫码NG抓取升降气缸缩回
AND 801.01  ; NG升降气缸1原位标志[0001.01]
AND 803.14  ; 扫码NG槽对射前光电有料标志[0003.14]
ORLD
LD D1013.13  ; 扫码NG放料拨料气缸伸出
AND 802.14  ; 料盒拨料气缸1到位标志[0002.14]
ORLD
LD D1013.14  ; 扫码NG放料拨料气缸缩回
AND 802.13  ; 料盒拨料气缸1原位标志[0002.13]
AND H20.10  ; 扫码NG抓取机构完成标志
ANDNOT H20.05  ; 扫码NG抓取机构忙绿标志
ORLD
LD D1013.15  ; 扫码NG抓取步序完成
AND P_Off
ORLD
AND D1016.00  ; 扫码NG抓取机构单步/自动循环运行
OUT D1012.01  ; 扫码NG抓取机构步进条件

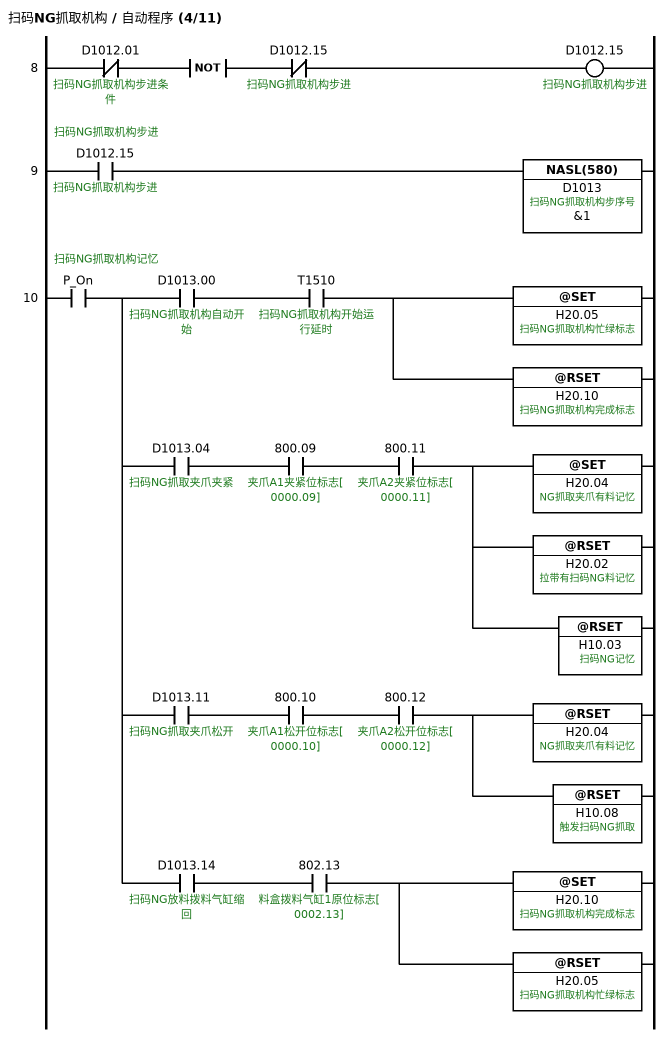
; rung 8
LDNOT D1012.01  ; 扫码NG抓取机构步进条件
NOT(520)
ANDNOT D1012.15  ; 扫码NG抓取机构步进
OUT D1012.15  ; 扫码NG抓取机构步进
; rung 9: 扫码NG抓取机构步进
LD D1012.15  ; 扫码NG抓取机构步进
NASL(580) D1013 &1  ; 扫码NG抓取机构步序号
; rung 10: 扫码NG抓取机构记忆
LD P_On
OUT TR0
AND D1013.00  ; 扫码NG抓取机构自动开始
AND T1510  ; 扫码NG抓取机构开始运行延时
@SET H20.05  ; 扫码NG抓取机构忙绿标志
@RSET H20.10  ; 扫码NG抓取机构完成标志
LD TR0
AND D1013.04  ; 扫码NG抓取夹爪夹紧
AND 800.09  ; 夹爪A1夹紧位标志[0000.09]
AND 800.11  ; 夹爪A2夹紧位标志[0000.11]
@SET H20.04  ; NG抓取夹爪有料记忆
@RSET H20.02  ; 拉带有扫码NG料记忆
@RSET H10.03  ; 扫码NG记忆
LD TR0
AND D1013.11  ; 扫码NG抓取夹爪松开
AND 800.10  ; 夹爪A1松开位标志[0000.10]
AND 800.12  ; 夹爪A2松开位标志[0000.12]
@RSET H20.04  ; NG抓取夹爪有料记忆
@RSET H10.08  ; 触发扫码NG抓取
LD TR0
AND D1013.14  ; 扫码NG放料拨料气缸缩回
AND 802.13  ; 料盒拨料气缸1原位标志[0002.13]
@SET H20.10  ; 扫码NG抓取机构完成标志
@RSET H20.05  ; 扫码NG抓取机构忙绿标志

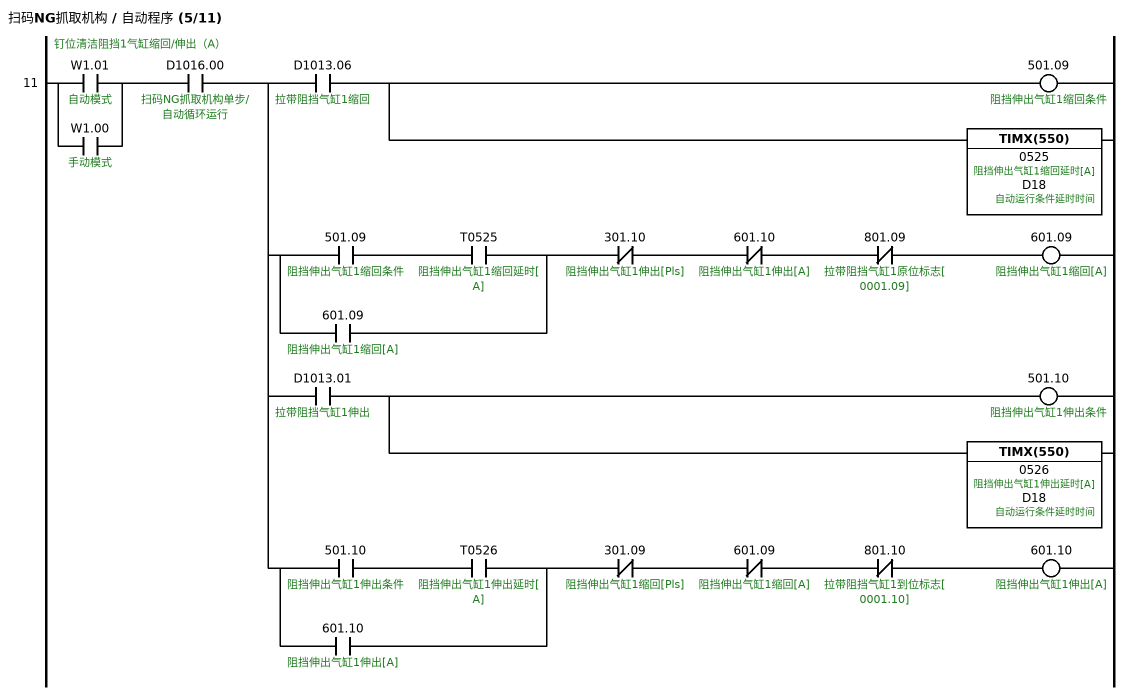
; rung 11: 钉位清洁阻挡1气缸缩回/伸出（A）
LD W1.01  ; 自动模式
OR W1.00  ; 手动模式
AND D1016.00  ; 扫码NG抓取机构单步/自动循环运行
OUT TR0
AND D1013.06  ; 拉带阻挡气缸1缩回
OUT 501.09  ; 阻挡伸出气缸1缩回条件
TIMX(550) 0525 D18  ; 自动运行条件延时时间, 阻挡伸出气缸1缩回延时[A]
LD TR0
LD 501.09  ; 阻挡伸出气缸1缩回条件
AND T0525  ; 阻挡伸出气缸1缩回延时[A]
OR 601.09  ; 阻挡伸出气缸1缩回[A]
ANDLD
ANDNOT 301.10  ; 阻挡伸出气缸1伸出[Pls]
ANDNOT 601.10  ; 阻挡伸出气缸1伸出[A]
ANDNOT 801.09  ; 拉带阻挡气缸1原位标志[0001.09]
OUT 601.09  ; 阻挡伸出气缸1缩回[A]
LD TR0
AND D1013.01  ; 拉带阻挡气缸1伸出
OUT 501.10  ; 阻挡伸出气缸1伸出条件
TIMX(550) 0526 D18  ; 自动运行条件延时时间, 阻挡伸出气缸1伸出延时[A]
LD TR0
LD 501.10  ; 阻挡伸出气缸1伸出条件
AND T0526  ; 阻挡伸出气缸1伸出延时[A]
OR 601.10  ; 阻挡伸出气缸1伸出[A]
ANDLD
ANDNOT 301.09  ; 阻挡伸出气缸1缩回[Pls]
ANDNOT 601.09  ; 阻挡伸出气缸1缩回[A]
ANDNOT 801.10  ; 拉带阻挡气缸1到位标志[0001.10]
OUT 601.10  ; 阻挡伸出气缸1伸出[A]

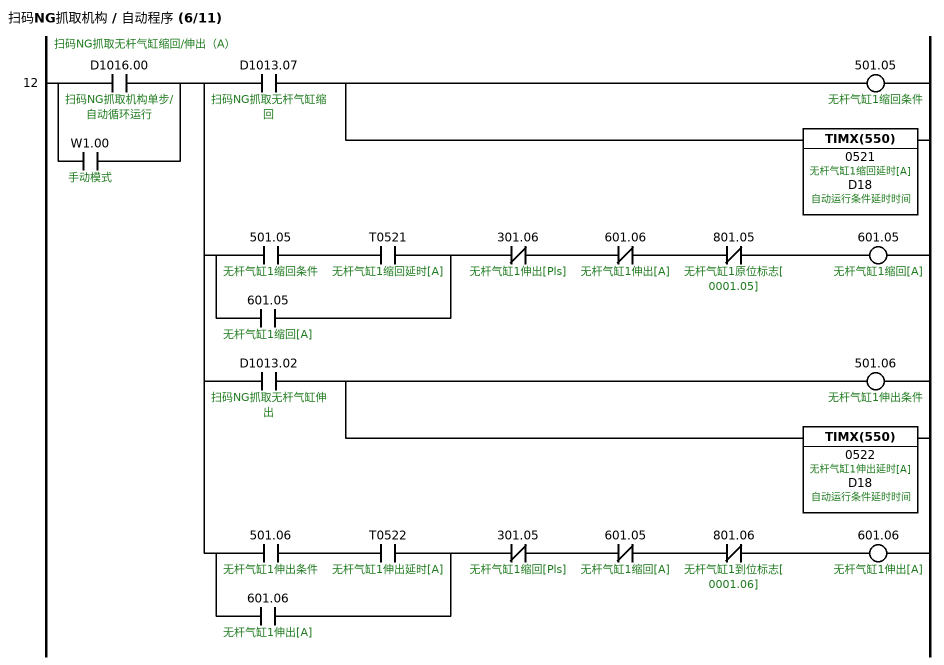
; rung 12: 扫码NG抓取无杆气缸缩回/伸出（A）
LD D1016.00  ; 扫码NG抓取机构单步/自动循环运行
OR W1.00  ; 手动模式
OUT TR0
AND D1013.07  ; 扫码NG抓取无杆气缸缩回
OUT 501.05  ; 无杆气缸1缩回条件
TIMX(550) 0521 D18  ; 自动运行条件延时时间, 无杆气缸1缩回延时[A]
LD TR0
LD 501.05  ; 无杆气缸1缩回条件
AND T0521  ; 无杆气缸1缩回延时[A]
OR 601.05  ; 无杆气缸1缩回[A]
ANDLD
ANDNOT 301.06  ; 无杆气缸1伸出[Pls]
ANDNOT 601.06  ; 无杆气缸1伸出[A]
ANDNOT 801.05  ; 无杆气缸1原位标志[0001.05]
OUT 601.05  ; 无杆气缸1缩回[A]
LD TR0
AND D1013.02  ; 扫码NG抓取无杆气缸伸出
OUT 501.06  ; 无杆气缸1伸出条件
TIMX(550) 0522 D18  ; 自动运行条件延时时间, 无杆气缸1伸出延时[A]
LD TR0
LD 501.06  ; 无杆气缸1伸出条件
AND T0522  ; 无杆气缸1伸出延时[A]
OR 601.06  ; 无杆气缸1伸出[A]
ANDLD
ANDNOT 301.05  ; 无杆气缸1缩回[Pls]
ANDNOT 601.05  ; 无杆气缸1缩回[A]
ANDNOT 801.06  ; 无杆气缸1到位标志[0001.06]
OUT 601.06  ; 无杆气缸1伸出[A]

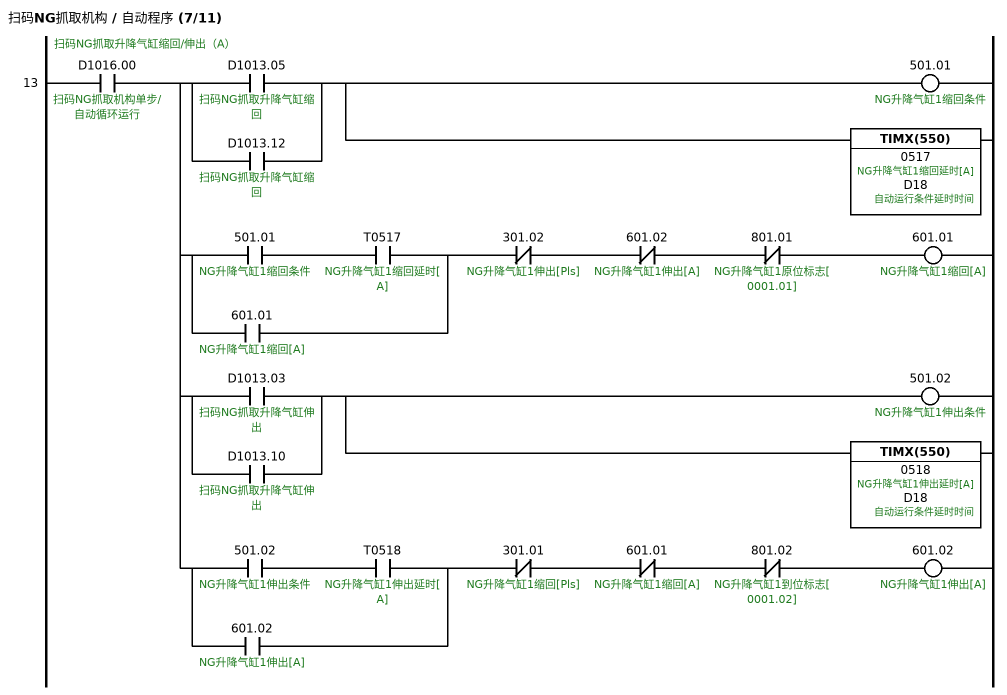
; rung 13: 扫码NG抓取升降气缸缩回/伸出（A）
LD D1016.00  ; 扫码NG抓取机构单步/自动循环运行
OUT TR0
LD D1013.05  ; 扫码NG抓取升降气缸缩回
OR D1013.12  ; 扫码NG抓取升降气缸缩回
ANDLD
OUT 501.01  ; NG升降气缸1缩回条件
TIMX(550) 0517 D18  ; 自动运行条件延时时间, NG升降气缸1缩回延时[A]
LD TR0
LD 501.01  ; NG升降气缸1缩回条件
AND T0517  ; NG升降气缸1缩回延时[A]
OR 601.01  ; NG升降气缸1缩回[A]
ANDLD
ANDNOT 301.02  ; NG升降气缸1伸出[Pls]
ANDNOT 601.02  ; NG升降气缸1伸出[A]
ANDNOT 801.01  ; NG升降气缸1原位标志[0001.01]
OUT 601.01  ; NG升降气缸1缩回[A]
LD TR0
LD D1013.03  ; 扫码NG抓取升降气缸伸出
OR D1013.10  ; 扫码NG抓取升降气缸伸出
ANDLD
OUT 501.02  ; NG升降气缸1伸出条件
TIMX(550) 0518 D18  ; 自动运行条件延时时间, NG升降气缸1伸出延时[A]
LD TR0
LD 501.02  ; NG升降气缸1伸出条件
AND T0518  ; NG升降气缸1伸出延时[A]
OR 601.02  ; NG升降气缸1伸出[A]
ANDLD
ANDNOT 301.01  ; NG升降气缸1缩回[Pls]
ANDNOT 601.01  ; NG升降气缸1缩回[A]
ANDNOT 801.02  ; NG升降气缸1到位标志[0001.02]
OUT 601.02  ; NG升降气缸1伸出[A]

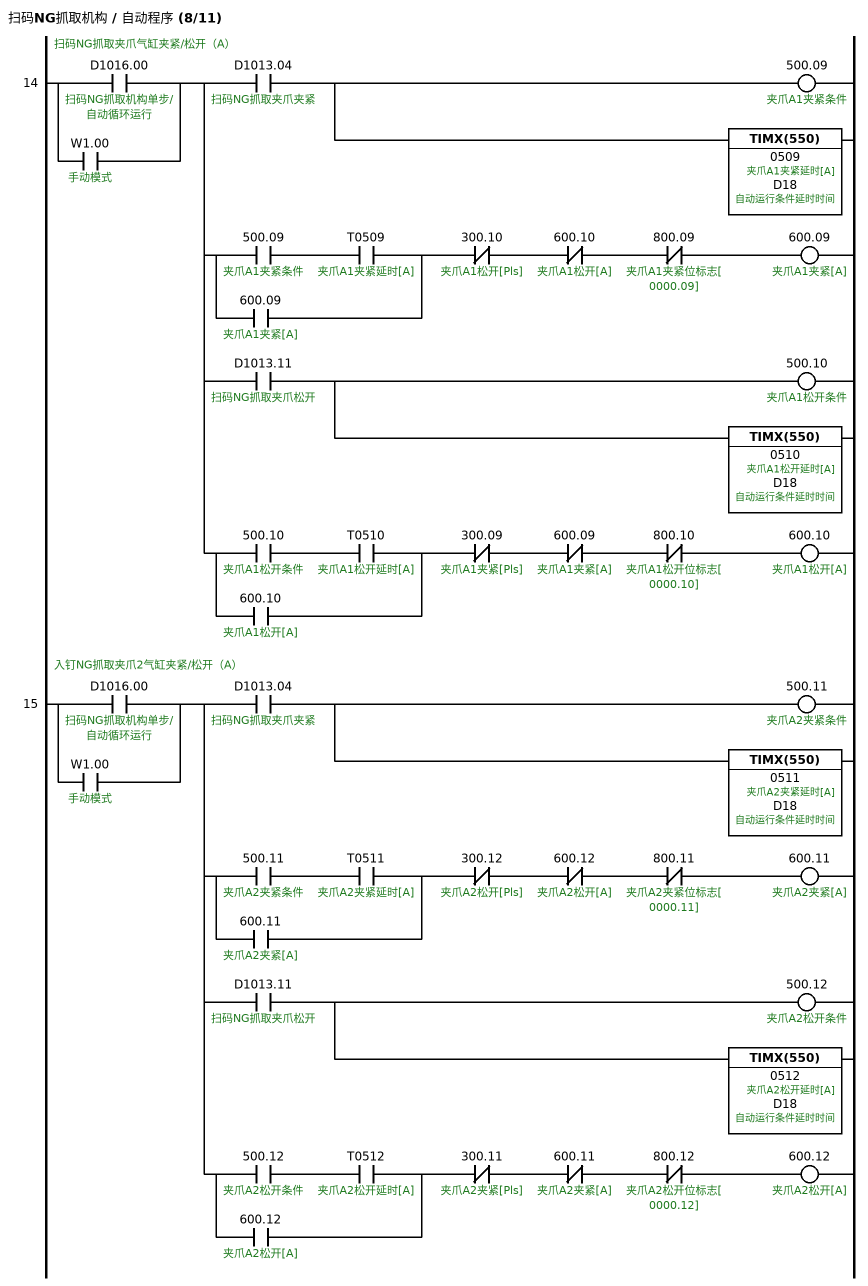
; rung 14: 扫码NG抓取夹爪气缸夹紧/松开（A）
LD D1016.00  ; 扫码NG抓取机构单步/自动循环运行
OR W1.00  ; 手动模式
OUT TR0
AND D1013.04  ; 扫码NG抓取夹爪夹紧
OUT 500.09  ; 夹爪A1夹紧条件
TIMX(550) 0509 D18  ; 自动运行条件延时时间, 夹爪A1夹紧延时[A]
LD TR0
LD 500.09  ; 夹爪A1夹紧条件
AND T0509  ; 夹爪A1夹紧延时[A]
OR 600.09  ; 夹爪A1夹紧[A]
ANDLD
ANDNOT 300.10  ; 夹爪A1松开[Pls]
ANDNOT 600.10  ; 夹爪A1松开[A]
ANDNOT 800.09  ; 夹爪A1夹紧位标志[0000.09]
OUT 600.09  ; 夹爪A1夹紧[A]
LD TR0
AND D1013.11  ; 扫码NG抓取夹爪松开
OUT 500.10  ; 夹爪A1松开条件
TIMX(550) 0510 D18  ; 自动运行条件延时时间, 夹爪A1松开延时[A]
LD TR0
LD 500.10  ; 夹爪A1松开条件
AND T0510  ; 夹爪A1松开延时[A]
OR 600.10  ; 夹爪A1松开[A]
ANDLD
ANDNOT 300.09  ; 夹爪A1夹紧[Pls]
ANDNOT 600.09  ; 夹爪A1夹紧[A]
ANDNOT 800.10  ; 夹爪A1松开位标志[0000.10]
OUT 600.10  ; 夹爪A1松开[A]
; rung 15: 入钉NG抓取夹爪2气缸夹紧/松开（A）
LD D1016.00  ; 扫码NG抓取机构单步/自动循环运行
OR W1.00  ; 手动模式
OUT TR0
AND D1013.04  ; 扫码NG抓取夹爪夹紧
OUT 500.11  ; 夹爪A2夹紧条件
TIMX(550) 0511 D18  ; 自动运行条件延时时间, 夹爪A2夹紧延时[A]
LD TR0
LD 500.11  ; 夹爪A2夹紧条件
AND T0511  ; 夹爪A2夹紧延时[A]
OR 600.11  ; 夹爪A2夹紧[A]
ANDLD
ANDNOT 300.12  ; 夹爪A2松开[Pls]
ANDNOT 600.12  ; 夹爪A2松开[A]
ANDNOT 800.11  ; 夹爪A2夹紧位标志[0000.11]
OUT 600.11  ; 夹爪A2夹紧[A]
LD TR0
AND D1013.11  ; 扫码NG抓取夹爪松开
OUT 500.12  ; 夹爪A2松开条件
TIMX(550) 0512 D18  ; 自动运行条件延时时间, 夹爪A2松开延时[A]
LD TR0
LD 500.12  ; 夹爪A2松开条件
AND T0512  ; 夹爪A2松开延时[A]
OR 600.12  ; 夹爪A2松开[A]
ANDLD
ANDNOT 300.11  ; 夹爪A2夹紧[Pls]
ANDNOT 600.11  ; 夹爪A2夹紧[A]
ANDNOT 800.12  ; 夹爪A2松开位标志[0000.12]
OUT 600.12  ; 夹爪A2松开[A]

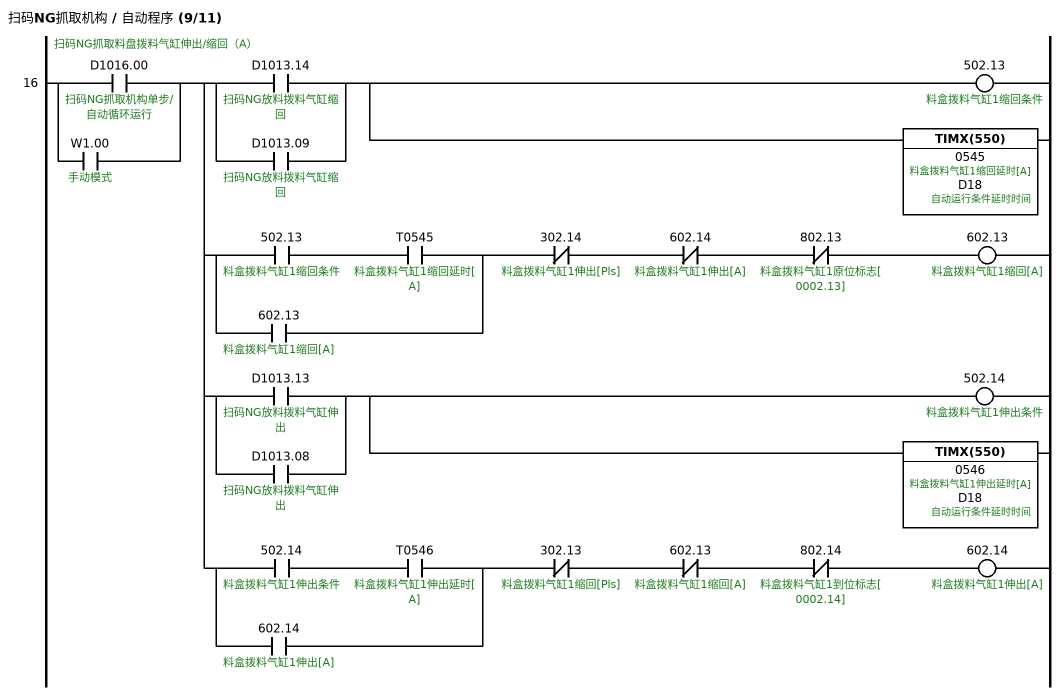
; rung 16: 扫码NG抓取料盘拨料气缸伸出/缩回（A）
LD D1016.00  ; 扫码NG抓取机构单步/自动循环运行
OR W1.00  ; 手动模式
OUT TR0
LD D1013.14  ; 扫码NG放料拨料气缸缩回
OR D1013.09  ; 扫码NG放料拨料气缸缩回
ANDLD
OUT 502.13  ; 料盒拨料气缸1缩回条件
TIMX(550) 0545 D18  ; 自动运行条件延时时间, 料盒拨料气缸1缩回延时[A]
LD TR0
LD 502.13  ; 料盒拨料气缸1缩回条件
AND T0545  ; 料盒拨料气缸1缩回延时[A]
OR 602.13  ; 料盒拨料气缸1缩回[A]
ANDLD
ANDNOT 302.14  ; 料盒拨料气缸1伸出[Pls]
ANDNOT 602.14  ; 料盒拨料气缸1伸出[A]
ANDNOT 802.13  ; 料盒拨料气缸1原位标志[0002.13]
OUT 602.13  ; 料盒拨料气缸1缩回[A]
LD TR0
LD D1013.13  ; 扫码NG放料拨料气缸伸出
OR D1013.08  ; 扫码NG放料拨料气缸伸出
ANDLD
OUT 502.14  ; 料盒拨料气缸1伸出条件
TIMX(550) 0546 D18  ; 自动运行条件延时时间, 料盒拨料气缸1伸出延时[A]
LD TR0
LD 502.14  ; 料盒拨料气缸1伸出条件
AND T0546  ; 料盒拨料气缸1伸出延时[A]
OR 602.14  ; 料盒拨料气缸1伸出[A]
ANDLD
ANDNOT 302.13  ; 料盒拨料气缸1缩回[Pls]
ANDNOT 602.13  ; 料盒拨料气缸1缩回[A]
ANDNOT 802.14  ; 料盒拨料气缸1到位标志[0002.14]
OUT 602.14  ; 料盒拨料气缸1伸出[A]

